Omron CX-Programmer project NewProject (CX-Programmer 9.75)

# PLC NewPLC1: CP2E-N N

## Global symbols (name address type ; comment)
0.00 BOOL  ; PROXY STOP KONVEYOR
0.01 BOOL  ; PROXY BOWL DISPENSER
0.02 BOOL  ; START BUTTON
100.00 BOOL  ; MOTOR BOWL DISPENSER
100.01 BOOL  ; MOTOR KONVEYOR 1
100.02 BOOL  ; MOTOR KONVEYOR
100.06 BOOL  ; MOTOR LINEAR ACTUATOR
10.02 BOOL  ; Cup Dispensed
200.00 BOOL  ; RELAY START
200.01 BOOL  ; RELAY START KONVEYOR
200.02 BOOL  ; RELAY ACTUATOR
200.03 BOOL  ; MOTOR BOWL
200.04 BOOL  ; RESET COUNTER
C000 BOOL  ; Mie Kering Count
C001 BOOL  ; Cup Count
D10 CHANNEL  ; OrderCount
D120 CHANNEL  ; Order Count (From PC)
D5 CHANNEL  ; OrderQty
D6 CHANNEL  ; Order1_Menu
D7 CHANNEL  ; Order2_Menu
D8 CHANNEL  ; Order3_Menu
T000 BOOL  ; TIMER ActuatorMie
T001 BOOL  ; Cycle1 finish
T002 BOOL  ; Reset Second Cup
T003 BOOL  ; Rst Third Cup State
T004 BOOL  ; On MODBUS
T005 BOOL  ; Interlock Linear Actuator retracted
T006 BOOL  ; Timer Boil Mie 1
T007 BOOL  ; Timer Pick Mie Kering 2
T008 BOOL  ; Timer Pick Mie Kering 3
T009 BOOL  ; Timer Boil Mie 2
T010 BOOL  ; Timer Boil Mie 3
W100.01 BOOL  ; MieKering_Ready
W100.02 BOOL  ; Cup_Ready
W100.03 BOOL  ; Boiling_Mie1
W100.04 BOOL  ; Boiling_Mie2
W100.05 BOOL  ; Boiling_Mie3
W100.06 BOOL  ; RebusMie1_Done
W100.07 BOOL  ; RebusMie2_Done
W100.08 BOOL  ; RebusMie3_Done
W100.09 BOOL  ; Start_PickMie2_ToRobot
W100.10 BOOL  ; Start_PickMie3_ToRobot
W100.11 BOOL  ; Order1Topping
W100.12 BOOL  ; Order2Topping
W100.13 BOOL  ; Order3Topping
W10.00 BOOL  ; RST
W10.01 BOOL  ; MieKering_Picked
W10.02 BOOL  ; Cup dispensed
W10.03 BOOL  ; CupReady
W11.00 BOOL  ; Delay 1sec Trigger
W120.00 BOOL  ; Finished Order From Robot
W12.00 BOOL  ; 1 Sec Delay
W1.00 BOOL  ; MieKering_Arrived
W1.01 BOOL  ; MieKering_Picked
W1.02 BOOL  ; Cup_Dropped
W2 CHANNEL  ; Multiple Order States
W20.00 BOOL  ; CheckOrder
W2.00 BOOL  ; ModbusStatus
W2.01 BOOL  ; TIMRST
W2.02 BOOL  ; 1stOrder Done
W2.03 BOOL  ; Second Cup Done
W2.04 BOOL  ; All Cup Done
W2.05 BOOL  ; ThirdCup
W2.06 BOOL  ; Second Cup
W2.07 BOOL  ; Third Cup Done
W2.08 BOOL  ; LockActuatorMie
W3 CHANNEL  ; Object Position States
W3.00 BOOL  ; StartRelay
W3.01 BOOL  ; MotorMie
W3.02 BOOL  ; Conveyor
W3.03 BOOL  ; Mie Sampe
W3.05 BOOL  ; BowlJatuh
W3.06 BOOL  ; Bowl Arrived
W3.07 BOOL  ; Second Cup
W5.00 BOOL  ; Start MODBUS
FB_MODBUSTCP_SERVER _CP2E003_ExecuteModTcpServer
Order1_Menu D110 CHANNEL
Order1_Topping1 D100 CHANNEL
Order1_Topping2 D101 CHANNEL
Order1_Topping3 D102 CHANNEL
Order2_Menu D111 CHANNEL
Order2_Topping1 D103 CHANNEL
Order2_Topping2 D104 CHANNEL
Order2_Topping3 D105 CHANNEL
Order3_Menu D112 CHANNEL
Order3_Topping1 D106 CHANNEL
Order3_Topping2 D107 CHANNEL
Order3_Topping3 D108 CHANNEL
Start_Order W100.00 BOOL

## Program MODBUS (cyclic task 0)
Local symbols
p_LT BOOL
p_eq BOOL
p_gt BOOL
p_lt BOOL

### Section MODBUS

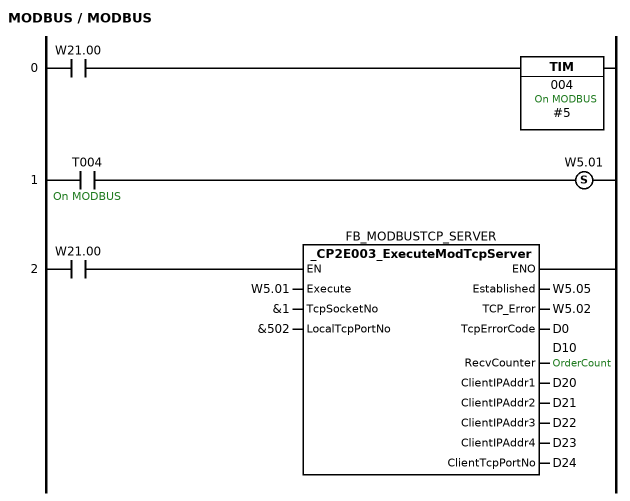
; rung 0
LD W21.00
TIM 004 #5  ; On MODBUS
; rung 1
LD T004  ; On MODBUS
SET W5.01
; rung 2
LD W21.00
CALL FB_MODBUSTCP_SERVER : _CP2E003_ExecuteModTcpServer (Execute := W5.01, TcpSocketNo := &1, LocalTcpPortNo := &502, Established => W5.05, TCP_Error => W5.02, TcpErrorCode => D0, RecvCounter => D10, ClientIPAddr1 => D20, ClientIPAddr2 => D21, ClientIPAddr3 => D22, ClientIPAddr4 => D23, ClientTcpPortNo => D24)  ; OrderCount

### Section Feeder_Main

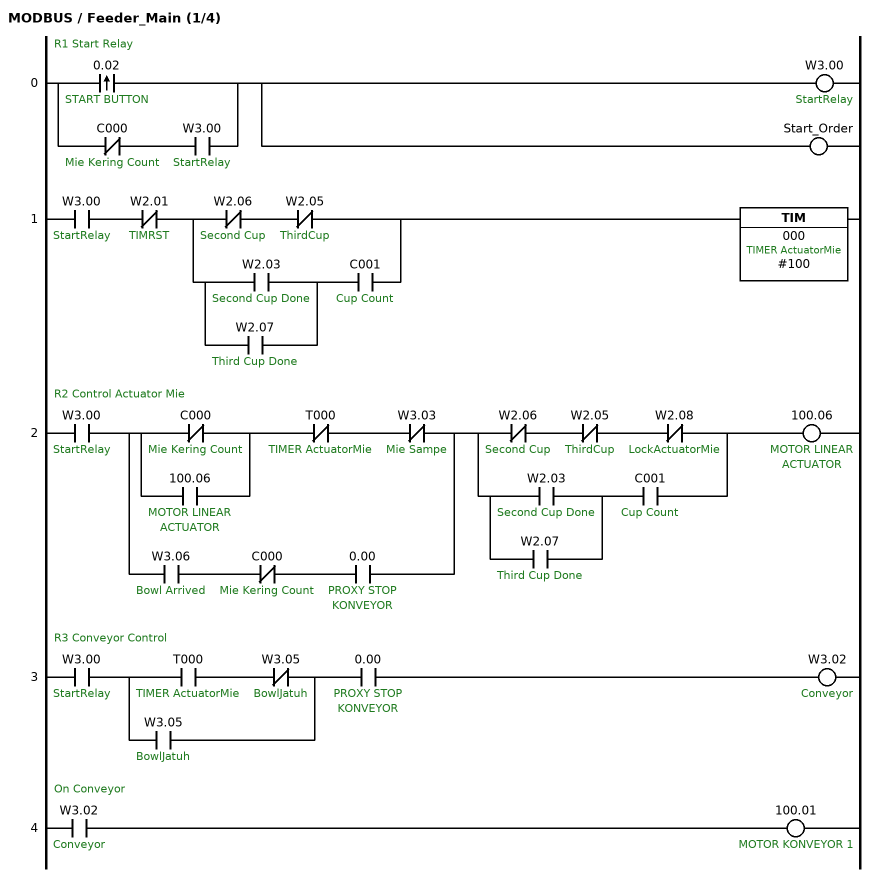
; rung 0: R1 Start Relay
@LD 0.02  ; START BUTTON
LDNOT C000  ; Mie Kering Count
AND W3.00  ; StartRelay
ORLD
OUT W3.00  ; StartRelay
OUT Start_Order
; rung 1
LD W3.00  ; StartRelay
ANDNOT W2.01  ; TIMRST
LDNOT W2.06  ; Second Cup
ANDNOT W2.05  ; ThirdCup
LD W2.03  ; Second Cup Done
OR W2.07  ; Third Cup Done
AND C001  ; Cup Count
ORLD
ANDLD
TIM 000 #100  ; TIMER ActuatorMie
; rung 2: R2 Control Actuator Mie
LD W3.00  ; StartRelay
LDNOT C000  ; Mie Kering Count
OR 100.06  ; MOTOR LINEAR ACTUATOR
ANDNOT T000  ; TIMER ActuatorMie
ANDNOT W3.03  ; Mie Sampe
LD W3.06  ; Bowl Arrived
ANDNOT C000  ; Mie Kering Count
AND 0.00  ; PROXY STOP KONVEYOR
ORLD
ANDLD
LDNOT W2.06  ; Second Cup
ANDNOT W2.05  ; ThirdCup
ANDNOT W2.08  ; LockActuatorMie
LD W2.03  ; Second Cup Done
OR W2.07  ; Third Cup Done
AND C001  ; Cup Count
ORLD
ANDLD
OUT 100.06  ; MOTOR LINEAR ACTUATOR
; rung 3: R3 Conveyor Control
LD W3.00  ; StartRelay
LD T000  ; TIMER ActuatorMie
ANDNOT W3.05  ; BowlJatuh
OR W3.05  ; BowlJatuh
ANDLD
AND 0.00  ; PROXY STOP KONVEYOR
OUT W3.02  ; Conveyor
; rung 4: On Conveyor
LD W3.02  ; Conveyor
OUT 100.01  ; MOTOR KONVEYOR 1

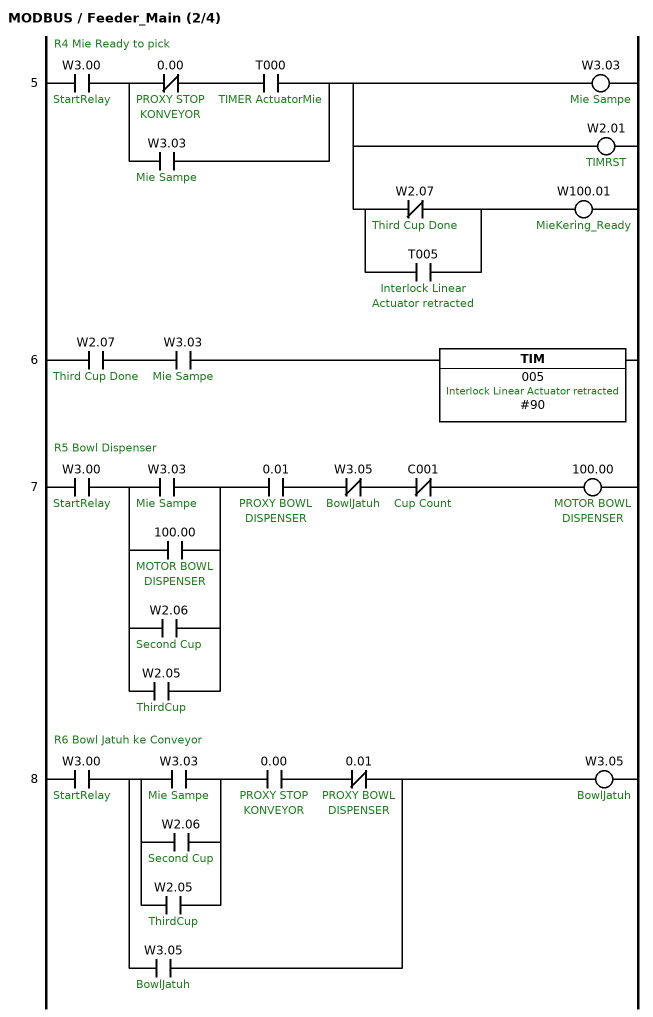
; rung 5: R4 Mie Ready to pick
LD W3.00  ; StartRelay
LDNOT 0.00  ; PROXY STOP KONVEYOR
AND T000  ; TIMER ActuatorMie
OR W3.03  ; Mie Sampe
ANDLD
OUT W3.03  ; Mie Sampe
OUT W2.01  ; TIMRST
LDNOT W2.07  ; Third Cup Done
OR T005  ; Interlock Linear Actuator retracted
ANDLD
OUT W100.01  ; MieKering_Ready
; rung 6
LD W2.07  ; Third Cup Done
AND W3.03  ; Mie Sampe
TIM 005 #90  ; Interlock Linear Actuator retracted
; rung 7: R5 Bowl Dispenser
LD W3.00  ; StartRelay
LD W3.03  ; Mie Sampe
OR 100.00  ; MOTOR BOWL DISPENSER
OR W2.06  ; Second Cup
OR W2.05  ; ThirdCup
ANDLD
AND 0.01  ; PROXY BOWL DISPENSER
ANDNOT W3.05  ; BowlJatuh
ANDNOT C001  ; Cup Count
OUT 100.00  ; MOTOR BOWL DISPENSER
; rung 8: R6 Bowl Jatuh ke Conveyor
LD W3.00  ; StartRelay
LD W3.03  ; Mie Sampe
OR W2.06  ; Second Cup
OR W2.05  ; ThirdCup
AND 0.00  ; PROXY STOP KONVEYOR
ANDNOT 0.01  ; PROXY BOWL DISPENSER
OR W3.05  ; BowlJatuh
ANDLD
OUT W3.05  ; BowlJatuh

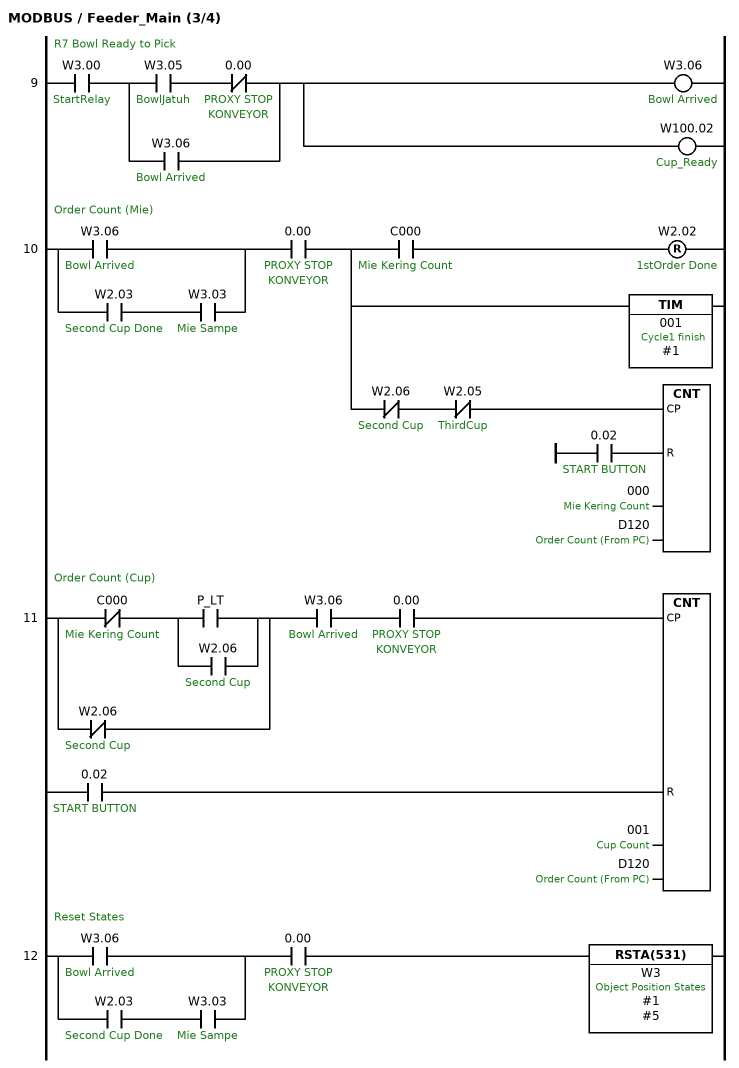
; rung 9: R7 Bowl Ready to Pick
LD W3.00  ; StartRelay
LD W3.05  ; BowlJatuh
ANDNOT 0.00  ; PROXY STOP KONVEYOR
OR W3.06  ; Bowl Arrived
ANDLD
OUT W3.06  ; Bowl Arrived
OUT W100.02  ; Cup_Ready
; rung 10: Order Count (Mie)
LD W3.06  ; Bowl Arrived
LD W2.03  ; Second Cup Done
AND W3.03  ; Mie Sampe
ORLD
AND 0.00  ; PROXY STOP KONVEYOR
OUT TR0
AND C000  ; Mie Kering Count
RSET W2.02  ; 1stOrder Done
LD TR0
TIM 001 #1  ; Cycle1 finish
ANDNOT W2.06  ; Second Cup
ANDNOT W2.05  ; ThirdCup
LD 0.02  ; START BUTTON
CNT 000 D120  ; Order Count (From PC), Mie Kering Count
; rung 11: Order Count (Cup)
LDNOT C000  ; Mie Kering Count
LD P_LT
OR W2.06  ; Second Cup
ANDLD
ORNOT W2.06  ; Second Cup
AND W3.06  ; Bowl Arrived
AND 0.00  ; PROXY STOP KONVEYOR
LD 0.02  ; START BUTTON
CNT 001 D120  ; Order Count (From PC), Cup Count
; rung 12: Reset States
LD W3.06  ; Bowl Arrived
LD W2.03  ; Second Cup Done
AND W3.03  ; Mie Sampe
ORLD
AND 0.00  ; PROXY STOP KONVEYOR
RSTA(531) W3 #1 #5  ; Object Position States

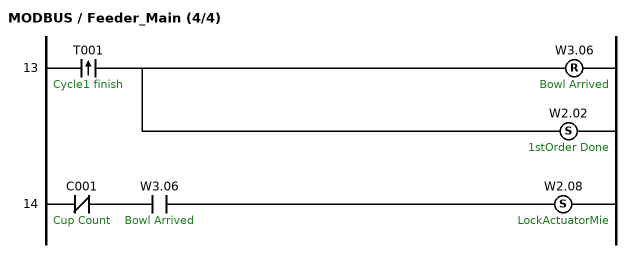
; rung 13
@LD T001  ; Cycle1 finish
RSET W3.06  ; Bowl Arrived
SET W2.02  ; 1stOrder Done
; rung 14
LDNOT C001  ; Cup Count
AND W3.06  ; Bowl Arrived
SET W2.08  ; LockActuatorMie

### Section Feeder_MultiOrder

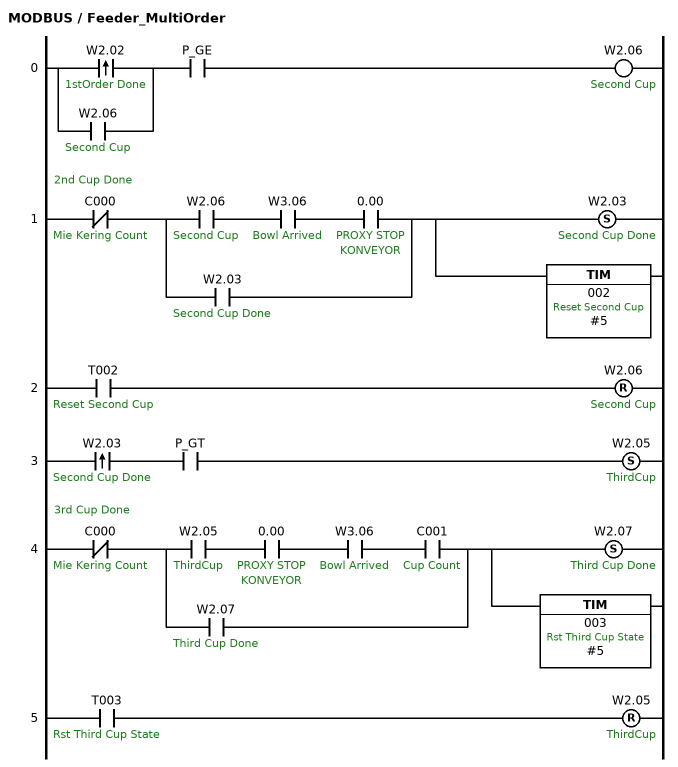
; rung 0
@LD W2.02  ; 1stOrder Done
OR W2.06  ; Second Cup
AND P_GE
OUT W2.06  ; Second Cup
; rung 1: 2nd Cup Done
LDNOT C000  ; Mie Kering Count
LD W2.06  ; Second Cup
AND W3.06  ; Bowl Arrived
AND 0.00  ; PROXY STOP KONVEYOR
OR W2.03  ; Second Cup Done
ANDLD
SET W2.03  ; Second Cup Done
TIM 002 #5  ; Reset Second Cup
; rung 2
LD T002  ; Reset Second Cup
RSET W2.06  ; Second Cup
; rung 3
@LD W2.03  ; Second Cup Done
AND P_GT
SET W2.05  ; ThirdCup
; rung 4: 3rd Cup Done
LDNOT C000  ; Mie Kering Count
LD W2.05  ; ThirdCup
AND 0.00  ; PROXY STOP KONVEYOR
AND W3.06  ; Bowl Arrived
AND C001  ; Cup Count
OR W2.07  ; Third Cup Done
ANDLD
SET W2.07  ; Third Cup Done
TIM 003 #5  ; Rst Third Cup State
; rung 5
LD T003  ; Rst Third Cup State
RSET W2.05  ; ThirdCup

### Section Order_Settings

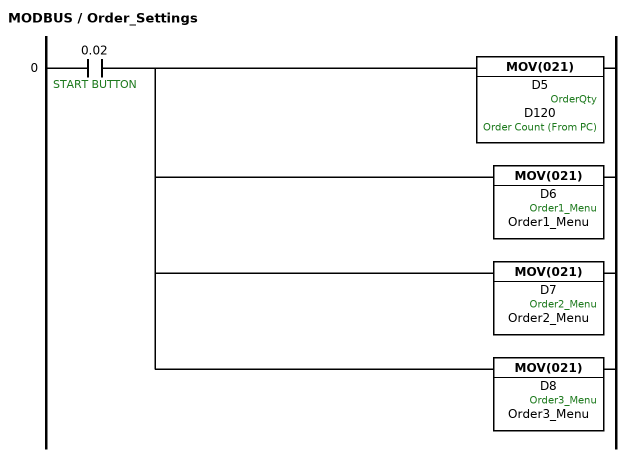
; rung 0
LD 0.02  ; START BUTTON
MOV(021) D5 D120  ; OrderQty, Order Count (From PC)
MOV(021) D6 Order1_Menu  ; Order1_Menu
MOV(021) D7 Order2_Menu  ; Order2_Menu
MOV(021) D8 Order3_Menu  ; Order3_Menu

### Section RESET_States

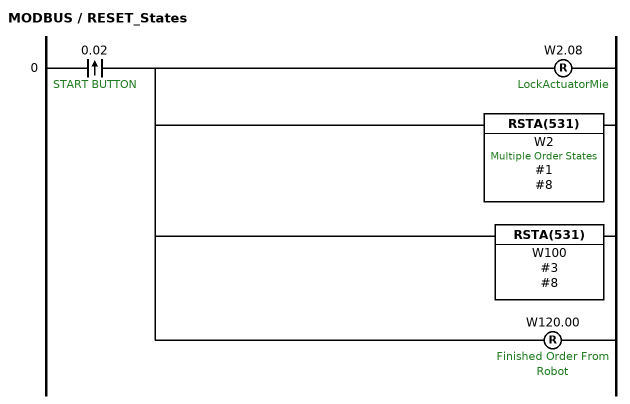
; rung 0
@LD 0.02  ; START BUTTON
RSET W2.08  ; LockActuatorMie
RSTA(531) W2 #1 #8  ; Multiple Order States
RSTA(531) W100 #3 #8
RSET W120.00  ; Finished Order From Robot

### Section Cooking_Process

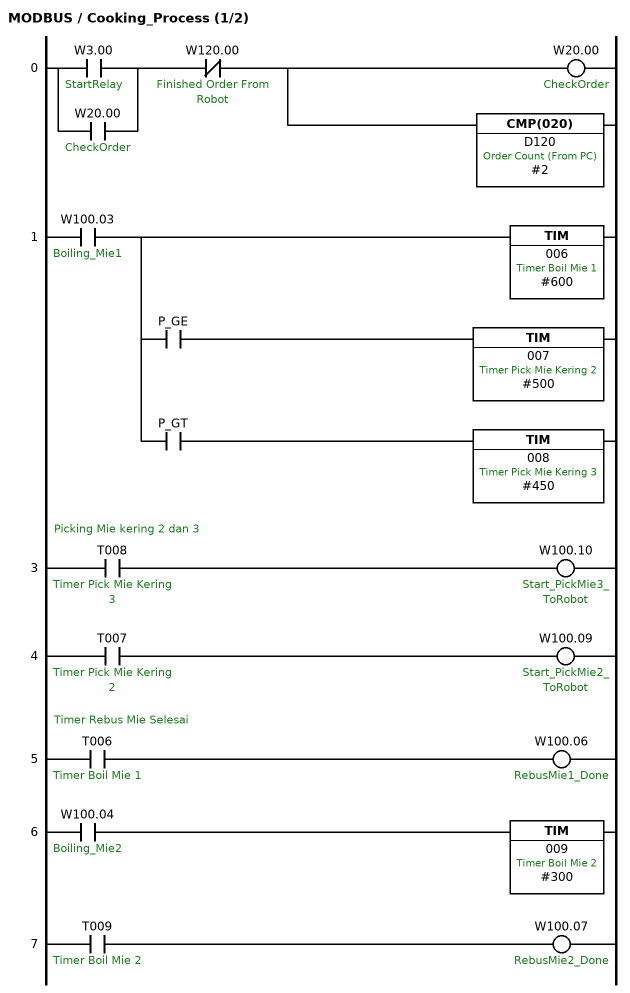
; rung 0
LD W3.00  ; StartRelay
OR W20.00  ; CheckOrder
ANDNOT W120.00  ; Finished Order From Robot
OUT W20.00  ; CheckOrder
CMP(020) D120 #2  ; Order Count (From PC)
; rung 1
LD W100.03  ; Boiling_Mie1
OUT TR0
TIM 006 #600  ; Timer Boil Mie 1
AND P_GE
TIM 007 #500  ; Timer Pick Mie Kering 2
LD TR0
AND P_GT
TIM 008 #450  ; Timer Pick Mie Kering 3
; rung 3: Picking Mie kering 2 dan 3
LD T008  ; Timer Pick Mie Kering 3
OUT W100.10  ; Start_PickMie3_ToRobot
; rung 4
LD T007  ; Timer Pick Mie Kering 2
OUT W100.09  ; Start_PickMie2_ToRobot
; rung 5: Timer Rebus Mie Selesai
LD T006  ; Timer Boil Mie 1
OUT W100.06  ; RebusMie1_Done
; rung 6
LD W100.04  ; Boiling_Mie2
TIM 009 #300  ; Timer Boil Mie 2
; rung 7
LD T009  ; Timer Boil Mie 2
OUT W100.07  ; RebusMie2_Done

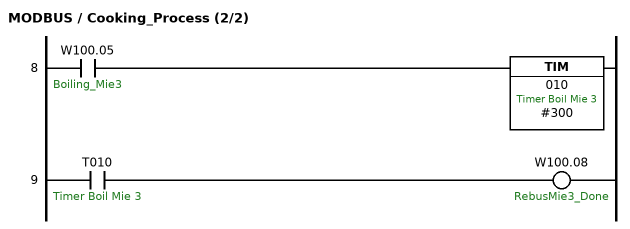
; rung 8
LD W100.05  ; Boiling_Mie3
TIM 010 #300  ; Timer Boil Mie 3
; rung 9
LD T010  ; Timer Boil Mie 3
OUT W100.08  ; RebusMie3_Done

### Section END
; rung 0
END(001)

## Function block _CP2E003_ExecuteModTcpServer (Omron library block, body left out)